FUNCTION_BLOCK AIS2_S_TO_STRING (* Composite FB for convert AIS2 to STRING *)
  (* Standard: 61499-2; Description: Copyright (c) 2024 HR Agrartechnik GmbH This program and the accompanying materials are made available under the terms of the Eclipse Public License 2.0 which is available at https://www.eclipse.org/legal/epl-2.0/ SPDX-License-Identifier: EPL-2.0 *)
  (* Version 1.0, 2026-09-12, Franz Höpfinger, HR Agrartechnik GmbH, Initial Version - Konvertierungsfamilie vervollstaendigt (analog zu AR2/AB2/AE2). *)
  PACKAGE adapter::conversion::bidirectional;
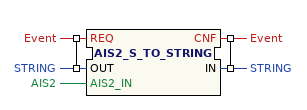
  EVENT_INPUT
    REQ WITH OUT; (* Request to Adapter *)
  END_EVENT
  EVENT_OUTPUT
    CNF WITH IN; (* Confirmation from Adapter *)
  END_EVENT
  VAR_INPUT
    OUT : STRING;
  END_VAR
  VAR_OUTPUT
    IN : STRING; (* Input data from Adapter *)
  END_VAR
  SOCKETS
    AIS2_IN : adapter::types::bidirectional::AIS2; (* Adapter Input *)
  END_SOCKETS
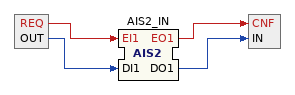
  EVENT_CONNECTIONS
    AIS2_IN.EO1 TO CNF;
    REQ TO AIS2_IN.EI1;
  END_CONNECTIONS
  DATA_CONNECTIONS
    AIS2_IN.DO1 TO IN;
    OUT TO AIS2_IN.DI1;
  END_CONNECTIONS
END_FUNCTION_BLOCK
